FUNCTION_BLOCK HydraulicValve
VAR_INPUT
	bvPosDir	: BOOL;
	bvNegDir	: BOOL;
	command		: REAL;
END_VAR
VAR
	rampTimeACC	: TIME;
	rampTimeDEC	: TIME;
	previousSolenoid	:	INT;	// -1 neg, 1 pos, 0 both min
	posDir	:	Solenoid();
	negDir	:	Solenoid(); 
	deltaCommand	:	REAL;
END_VAR
VAR_OUTPUT
	OutPosDir : REAL := 0 ;	// Výstup v daném směru [mA]
	OutNegDir : REAL := 0 ;	// Výstup v daném směru [mA]
END_VAR

IF NOT(generalVariable.staus.bBussy) THEN
	previousSolenoid := howIsActive();
	IF ((command - OutPosDir-OutNegDir) <> 0) THEN
		IF (previousSolenoid * command > 0) THEN
			// na istom solenoidu
			callSolenoid(posDirB := bvPosDir, desPosition := ABS(command));
			ELSIF (previousSolenoid * command < 0) THEN
				//postoji prelaz
				callSolenoid(posDirB := bvPosDir, desPosition := 0);
				ELSE
					// error there is no allowed direction		
					generalVariable.staus.Standstill := TRUE;			
					END_IF;
			END_IF;
	END_IF;

METHOD PRIVATE callSolenoid
VAR_INPUT
	posDirB	:	BOOL;
	desPosition	:	REAL;
END_VAR
IF posDirB THEN
	posDir(activeSolenoid := posDirB, desiredPosition := desPosition);
	ELSE
		negDir(activeSolenoid := posDirB, desiredPosition := desPosition);
		END_IF;
END_METHOD

METHOD howIsActive :INT
VAR_INPUT
END_VAR
IF posDir.activeSolenoid THEN
	howIsActive := 1;
	generalVariable.staus.OutPosDirProc := command;
	generalVariable.staus.OutNegDirProc := 0;
	ELSIF negDir.activeSolenoid THEN
		howIsActive := -1;
		generalVariable.staus.OutPosDirProc := 0;
		generalVariable.staus.OutNegDirProc := command;
		ELSE
			howIsActive := 0;
			END_IF;
END_METHOD

METHOD PRIVATE RampTimeNeg : REAL
IF bvPosDir THEN
	rampTimeACC:= INT_TO_TIME(REAL_TO_INT(generalVariable.conParammetr.CurNegDirMax/generalVariable.conParammetr.RampNegDirUp));
	ELSE
		rampTimeDEC := INT_TO_TIME(REAL_TO_INT(generalVariable.conParammetr.CurNegDirMin/generalVariable.conParammetr.RampNegDirDown));
		END_IF;
END_METHOD

METHOD PRIVATE RampTimePos : REAL
IF bvPosDir THEN
	rampTimeACC := INT_TO_TIME(REAL_TO_INT(generalVariable.conParammetr.CurPosDirMax/generalVariable.conParammetr.RampPosDirUp));
	ELSE
		rampTimeDEC := INT_TO_TIME(REAL_TO_INT(generalVariable.conParammetr.CurPosDirMin/generalVariable.conParammetr.RampPosDirDown));
		END_IF;
END_METHOD

END_FUNCTION_BLOCK

(* stored: Version 1.1.0.1, ProductVersion 3.1.4024.12
   POU HydraulicValve: Id {52b97062-b094-41f2-9637-f563a04dcc55}, SpecialFunc None
   Method callSolenoid: Id {046924e7-1f03-422e-ac99-a6cc7cb22e47}
   Method howIsActive: Id {e3d729e3-05dd-414f-8828-4f1662c60e24}
   Method RampTimeNeg: Id {2afb1cac-dc67-43e1-8d1a-3c7ce10f6c11}
   Method RampTimePos: Id {d7afd6bf-2929-4b9b-8946-24d995302043} *)
